{attribute 'linkalways'} 
{attribute 'no_explicit_call' := 'This FB is a CLASS and must be accessed using methods or properties'}
{attribute 'enable_dynamic_creation'}
FUNCTION_BLOCK InvalidArrayIndexDeserializationError EXTENDS Error
VAR
	index : UDINT;
END_VAR

PROPERTY PUBLIC ErrorType : T_MAXSTRING
GET
ErrorType := 'INVALID_ARRAY_INDEX_DESERIALIZATION_ERROR';
END_GET
END_PROPERTY

METHOD FB_init : BOOL
VAR_INPUT
	bInitRetains : BOOL; // if TRUE, the retain variables are initialized (warm start / cold start)
	bInCopyCode : BOOL;  // if TRUE, the instance afterwards gets moved into the copy code (online change)
	Index : UDINT;
END_VAR
this^.index := Index;
END_METHOD

PROPERTY PUBLIC Message : T_MAXSTRING
GET
Message := CONCAT('Deserialization Failed, Array Index Out Of Bounds ', UDINT_TO_STRING(index));
END_GET
END_PROPERTY

END_FUNCTION_BLOCK

(* stored: Version 1.1.0.1, ProductVersion 3.1.4024.13
   POU InvalidArrayIndexDeserializationError: Id {11d6e6a2-6083-06be-2e22-e7e6f3e01f83}, SpecialFunc None
   Folder Constructor: Id {4a9af5f6-0ac3-0fa8-16f8-1f034c004d45}
   Property ErrorType: Id {0708fdf4-b5ef-0898-0b51-0d2437b5653d}
   Get Get: Id {9a2adaf5-40ca-0b12-21ab-f730de041c2b}
   Method FB_init: Id {7be0ce88-ac66-056b-0a72-78f1a7b988e2}
   Property Message: Id {598bfc12-9466-0ec5-1108-f69ee4c1b1af}
   Get Get: Id {0051b229-1263-0621-0178-3bb0bf18eecf} *)
